PROGRAM MAIN
VAR
	fbSimpleUpload 		: FB_SimpleUpload;
	fbSimpleDownload 	: FB_SimpleDownload;
	fbManualOperation 	: FB_ManualOperation;
END_VAR

fbManualOperation();
fbSimpleUpload();
fbSimpleDownload();

END_PROGRAM

(* stored: Version 1.1.0.1, ProductVersion 3.1.4026.8
   POU MAIN: Id {0a1a5817-b9f5-41e5-ac48-866a84c77eb8}, SpecialFunc None *)
